// TwinCAT 3 PLC project PLC_IotBase_Test
// ProgramVersion: 3.1.4020.4
// libraries:
//   Tc2_Standard, * (Beckhoff Automation GmbH)
//   Tc2_System, * (Beckhoff Automation GmbH)
//   Tc2_Utilities, * (Beckhoff Automation GmbH)
//   Tc3_DynamicMemory, * (Beckhoff Automation GmbH)
//   Tc3_JsonXml, * (Beckhoff Automation GmbH)
//   Tc3_Module, * (Beckhoff Automation GmbH)
//   Tc3_IotBase,3.1.8.3,Beckhoff Automation GmbH
// project tree:
//   / PlcTask.TcTTO
//   POUs/ FB_TestHTTPLegacy.TcPOU, FB_TestHTTP.TcPOU, FB_TestHTTP_Delete.TcPOU, FB_TestHTTP_Get2.TcPOU, FB_TestHTTP_Trace.TcPOU, FB_TestHTTP_Head.TcPOU, FB_TestHTTP_Connect.TcPOU, FB_TestHTTP_Post.TcPOU, FB_TestHTTP_Get.TcPOU, FB_TestHTTP_Put.TcPOU, FB_TestHTTP_Patch.TcPOU, FB_TestHTTP_Options.TcPOU, FB_TestMqtt.TcPOU, MAIN.TcPOU
// real-time tasks:
//   TASK PlcTask: cycle T#10ms, priority 20, ADS port 350

CONFIGURATION PLC_IotBase_Test
    RESOURCE PLC ON TwinCAT3
        TASK PlcTask(INTERVAL := T#10ms, PRIORITY := 20);
        PROGRAM MAIN WITH PlcTask : MAIN;
    END_RESOURCE
END_CONFIGURATION

// ---- POUs/MAIN.TcPOU
PROGRAM MAIN
VAR
	i : INT;
	bTestMqtt : BOOL;
	fbMqtt : FB_TestMqtt;
	bTestHttp : BOOL := TRUE;
	fbHttp : FB_TestHTTP;
	
END_VAR

i := i + 1;

IF bTestMqtt THEN
	fbMqtt();	
END_IF
IF bTestHttp THEN
	fbHttp();	
END_IF

END_PROGRAM

// ---- POUs/FB_TestMqtt.TcPOU
{attribute 'c++_compatible'}
FUNCTION_BLOCK FB_TestMqtt EXTENDS FB_IotMqttClient
VAR
	hrLastErrorCode : HRESULT;
	bGet : BOOL := TRUE;
	bSetParameter : BOOL := TRUE;
	bConnect : BOOL := TRUE;
	bResetQueue : BOOL;
	sWillPayload : STRING := 'Ich bin dann mal weg.';
	
(* publish *)
	i: INT;
	m : USINT;
	sStr : STRING;
	sTopic1 : STRING(999) := 'test';
	{attribute 'TcEncoding':='UTF-8'}
	sPayload1Wr : STRING := 'Hello world!'; // := STRINGLITERAL_TO_UTF8('Hello world! (üöä)');
	sTopic2 : STRING(999) := '123456789012345678901234567890123456789012345678901234567890123456789012345678901234567890'; // 90 character long
	{attribute 'TcEncoding':='UTF-8'}
	sPayload2Wr : STRING := 'too long?';

(* subscribe *)
	bSubscribed: BOOL;
	{attribute 'TcEncoding':='UTF-8'}
	sPayload1Rd : STRING;
	{attribute 'TcEncoding':='UTF-8'}
	sPayload2Rd : STRING;
	sLastTopic : T_MaxString;
	fbMessageQueue : FB_IotMqttMessageQueue;
	fbMessage : FB_IotMqttMessage;
END_VAR

IF bSetParameter THEN
	bSetParameter := FALSE;
//	SUPER^.sClientId := 'MyTcMqttClient';
	SUPER^.sTopicPrefix := '';
//	SUPER^.sHostName := '172.17.62.85'; //'ba-tradeshows.cloudapp.net', // 'iot.beckhoff.com';
	SUPER^.nHostPort := 1883;
	SUPER^.sUserName := '';
	SUPER^.sUserPassword := '';
	SUPER^.sTopicPrefix := '';
	SUPER^.stTLS.sCA := ''; 
	SUPER^.nKeepAlive := 5;
	
	SUPER^.stWill.sTopic := 'test';
	SUPER^.stWill.pPayload := ADR(sWillPayload);
	SUPER^.stWill.nPayloadSize :=  LEN2(ADR(sWillPayload))+1;
(*
	SUPER^.sTopicPrefix := '';
	SUPER^.sHostName := 'ba-messagebroker.westeurope.cloudapp.azure.com'; // 'localhost'; //'ba-tradeshows.cloudapp.net', // 'iot.beckhoff.com';
	SUPER^.nHostPort := 8883; // 1883;
	SUPER^.sUserName := 'IotAnalytics';
	SUPER^.sUserPassword := '123456';
	SUPER^.sTopicPrefix := 'Beckhoff/Internal/IotAnalytics/';
	SUPER^.stTLS.sCA := 'C:\Projects\IotComm\CA\ca.crt'; // ''; 
*)
	SUPER^.ipMessageQueue := fbMessageQueue;
END_IF

Execute(bConnect);
IF bError THEN
	hrLastErrorCode := hrErrorCode;
END_IF

IF eConnectionState <> ETcIotMqttClientState.MQTT_ERR_NO_CONN THEN
	bConnected := bConnected; // for debugging purposes
END_IF

IF fbMessageQueue.nQueuedMessages > 0 AND bGet THEN
	IF fbMessageQueue.Dequeue(fbMessage) THEN
		IF fbMessage.CompareTopic(sTopic1) THEN
			fbMessage.GetPayload(ADR(sPayload1Rd), SIZEOF(sPayload1Rd), FALSE);
		ELSIF fbMessage.CompareTopic(sTopic2) THEN
			fbMessage.GetPayload(ADR(sPayload2Rd), SIZEOF(sPayload2Rd), FALSE);
		END_IF
	END_IF
END_IF

IF bResetQueue THEN
	bResetQueue := FALSE;
	fbMessageQueue.ResetQueue();
END_IF

IF bConnected THEN
	// subscrive
	IF NOT bSubscribed THEN
		IF Subscribe(sTopic1, 0) AND Subscribe(sTopic2, 0) THEN
			bSubscribed := TRUE;
		ELSE
			hrLastErrorCode := hrErrorCode;
		END_IF
	END_IF
	
	// publish
	i := i + 1;
	IF i = 100 THEN
		m := m + 1;
		sStr := CONCAT('Hello World! (üöä) - ', INT_TO_STRING(m));
		STRING_TO_UTF8(ADR(sPayload1Wr), ADR(sStr), SIZEOF(sPayload1Wr) );
		Publish(sTopic1, ADR(sPayload1Wr), INT_TO_UDINT(LEN(sPayload1Wr)+1), TcIotMqttQos.ExactlyOnceDelivery, FALSE, FALSE);
		IF bError THEN
			hrLastErrorCode := hrErrorCode;
		END_IF
	ELSIF i = 200 THEN
		sPayload1Wr := 'All right?';
		Publish(sTopic1, ADR(sPayload1Wr), INT_TO_UDINT(LEN(sPayload1Wr)+1), 0, FALSE, FALSE);
		IF bError THEN
			hrLastErrorCode := hrErrorCode;
		END_IF
		Publish(sTopic2, ADR(sPayload2Wr), INT_TO_UDINT(LEN(sPayload2Wr)+1), 0, FALSE, FALSE);
		IF bError THEN
			hrLastErrorCode := hrErrorCode;
		END_IF
		i := 0;
	END_IF	
END_IF

{attribute 'c++_compatible'}
{attribute 'signature_flag' := '33554688'}
{attribute 'pack_mode' := '4'}
{attribute 'show'}
{attribute 'minimal_input_size' := '4'}
{attribute 'checksuperglobal'}
METHOD OnMqttMessage : HRESULT
VAR_IN_OUT CONSTANT
	topic	: STRING;
END_VAR
VAR_INPUT
	payload	: PVOID;
	length	: UDINT;
	qos	: TcIotMqttQos;
	repeated	: BOOL;
END_VAR
nMessagesRcv := nMessagesRcv + 1;

STRNCPY( ADR(sLastTopic), ADR(topic), SIZEOF(sLastTopic) );

IF sLastTopic = CONCAT(SUPER^.sTopicPrefix, sTopic1) THEN
	MEMCPY(ADR(sPayload1Rd), payload, MIN(length, DINT_TO_UDINT(SIZEOF(sPayload1Rd))));
ELSIF sLastTopic = CONCAT(SUPER^.sTopicPrefix, sTopic2) THEN
	MEMCPY(ADR(sPayload2Rd), payload, MIN(length, DINT_TO_UDINT(SIZEOF(sPayload2Rd))));
END_IF

OnMqttMessage := S_OK;
END_METHOD

END_FUNCTION_BLOCK

// ---- POUs/FB_TestHTTP.TcPOU
FUNCTION_BLOCK FB_TestHTTP
VAR
	fbClient : FB_IotHttpClient;
	fbRequest: FB_IotHttpRequest;
	fbHeader: FB_IotHttpHeaderFieldMap;
	state : UDINT;
	timeout : UDINT :=10000;
	port : UINT:= 443;
		
	//http://jsonplaceholder.typicode.com/todos/1
	sHostName  : STRING(255) :='jsonplaceholder.typicode.com';
	sCA : STRING(255) := ''; // 'C:\TwinCAT\3.1\Target\Certificates\cloudflare.cer' tls vesrion 1.3 not supported

	fbMqtt_Post: FB_TestHTTP_Post;
	fbMqtt_Get: FB_TestHTTP_Get;
	fbMqtt_Get2: FB_TestHTTP_Get2;	
	fbMqtt_Put: FB_TestHTTP_Put;
	fbMqtt_Patch: FB_TestHTTP_Patch;
	fbMqtt_Trace: FB_TestHTTP_Trace;	
	fbMqtt_Head: FB_TestHTTP_Head;
	fbMqtt_Options: FB_TestHTTP_Options;
	fbMqtt_Delete: FB_TestHTTP_Delete;
	fbMqtt_Connect: FB_TestHTTP_Connect;			
END_VAR

CASE state OF
0:
	fbClient.nConnectTimeout := timeout;
	fbClient.sHostName := sHostName;
	fbClient.bKeepAlive := TRUE;
	IF LEN(STR:=sCA) = 0 THEN
		port:= 80;	
	END_IF
	fbClient.nHostPort := port;
	IF port = 443 THEN
		fbClient.stTLS.sCA :=  sCA;
	END_IF			
	fbHeader.AddField(sField:='MyField', sValue:='MyFieldValue', bAppendValue:= FALSE);
	IF fbClient.bConfigured THEN
		fbClient.Disconnect();
	END_IF	 
	state:=1;
1:	
	IF fbClient.bConfigured THEN 
		fbMqtt_Get(fbClient:=fbClient);
		fbMqtt_Get2(fbClient:=fbClient);
		fbMqtt_Post(fbClient:=fbClient);
		fbMqtt_Put(fbClient:=fbClient);
		fbMqtt_Patch(fbClient:=fbClient);
		fbMqtt_Trace(fbClient:=fbClient);
		fbMqtt_Head(fbClient:=fbClient);
		fbMqtt_Options(fbClient:=fbClient);
		fbMqtt_Delete(fbClient:=fbClient);
		fbMqtt_Connect(fbClient:=fbClient);
	END_IF  	
END_CASE
fbClient.Execute();

END_FUNCTION_BLOCK

// ---- POUs/FB_TestHTTP_Post.TcPOU
FUNCTION_BLOCK FB_TestHTTP_Post
VAR_INPUT
	fbClient : REFERENCE TO FB_IotHttpClient;
END_VAR
VAR	
	fbRequest: FB_IotHttpRequest;
	fbJson: FB_JsonDomParser;
	bSend : BOOL;
	bContinuous : BOOL;
	state : UDINT;
	
	RisingEdge		: R_TRIG;
	sJson: STRING(1024);
	sContent: STRING(1024);	
	
	bJsonRes : BOOL;
	jsonDoc    : SJsonValue;
	jsonVal    : SJsonValue;
		
	reqCount : UDINT;		
	invResCount : UDINT := 0;
	invResValCount : UDINT := 0;
	resVal:STRING;
	nResCnt : UDINT;
	nErrCnt1 : UDINT;
	nErrCnt2 : UDINT;
		
	valOkCount: UDINT;
	
	//http://jsonplaceholder.typicode.com/todos/1
	sUri: STRING(255) := '/posts';
	eRequestType : ETcIotHttpRequestType := ETcIotHttpRequestType.HTTP_POST;		
END_VAR

RisingEdge( CLK:= bSend );
CASE state OF
0:		
	IF fbClient.bConfigured AND (RisingEdge.Q OR bContinuous) THEN 
		fbJson.NewDocument();
		jsonDoc := fbJson.GetDocumentRoot();
		fbJson.AddStringMember(jsonDoc, 'title', 'test1');
		fbJson.AddStringMember(jsonDoc, 'body', 'test2');
		fbJson.AddUintMember(jsonDoc, 'userId', reqCount);
		IF fbRequest.SendJsonDomRequest(sUri:=sUri, fbClient:=fbClient, eRequestType:=eRequestType, fbJson, 0) THEN				
			state := 1;
			reqCount:=reqCount+1;
		END_IF					
	END_IF
1:
	IF NOT fbRequest.bBusy THEN
			IF NOT fbRequest.bError THEN				 
				jsonDoc := fbRequest.GetJsonDomContent(fbJson);				
				IF  jsonDoc <> 0 THEN
					bJsonRes := TRUE;
					fbJson.CopyDocument(sJson, SIZEOF(sJson));
				ELSE
					bJsonRes := FALSE;
				END_IF					
				fbRequest.GetContent(pContent:=ADR(sContent), nContentSize:=SIZEOF(sContent), bSetNullTermination:=TRUE);	
				IF fbRequest.nStatusCode >= 200 AND fbRequest.nStatusCode < 300 THEN
					IF bJsonRes THEN
						IF fbJson.HasMember(jsonDoc, 'userId')  THEN
							jsonVal := fbJson.FindMember(jsonDoc, 'userId');
							IF fbJson.GetUint(jsonVal)+1 = reqCount THEN
								valOkCount:=valOkCount+1;
							ELSE
								invResValCount:=invResValCount+1;
							END_IF
						ELSE 
							invResCount:=invResCount+1;	
						END_IF
					ELSE
						invResCount:=invResCount+1;
					END_IF					
					nResCnt:=nResCnt+1;
				ELSE
					nErrCnt1:=nErrCnt1+1;					
				END_IF				
			ELSE
				nErrCnt2:=nErrCnt2+1;
			END_IF
			state :=0;				
	END_IF  	
END_CASE
fbClient.Execute();

END_FUNCTION_BLOCK

// ---- POUs/FB_TestHTTP_Get.TcPOU
FUNCTION_BLOCK FB_TestHTTP_Get
VAR_INPUT
	fbClient : REFERENCE TO FB_IotHttpClient;
END_VAR
VAR
	
	fbRequest: FB_IotHttpRequest;
	fbJson: FB_JsonDomParser;
	bSend : BOOL;
	bContinuous : BOOL;
	state : UDINT;
	
	RisingEdge		: R_TRIG;
	
	sJson: STRING(300);		
	sContent1: STRING(291);
	bGetContent1 : BOOL;
	nContent1 : UDINT;
	
	bJsonRes : BOOL;
	jsonDoc    : SJsonValue;
	jsonVal    : SJsonValue;
		
	reqCount : UDINT;		
	invResCount : UDINT := 0;
	invResValCount : UDINT := 0;
	resVal:STRING;
	nResCnt : UDINT;
	nErrCnt1 : UDINT;
	nErrCnt2 : UDINT;
		
	valOkCount: UDINT;	
	
	sUri: STRING(255) := '/posts';
	eRequestType : ETcIotHttpRequestType := ETcIotHttpRequestType.HTTP_Get;		
END_VAR

RisingEdge( CLK:= bSend );
CASE state OF
0:	
	IF fbClient.bConfigured AND (RisingEdge.Q OR bContinuous) THEN 
		IF fbRequest.SendRequest(sUri:=sUri, fbClient:=fbClient, eRequestType:=eRequestType, 0, 0, 0) THEN				
			state := 1;
			reqCount:=reqCount+1;
		END_IF					
	END_IF
1:
	IF NOT fbRequest.bBusy THEN
			IF NOT fbRequest.bError THEN				 
				jsonDoc := fbRequest.GetJsonDomContent(fbJson);
				IF  jsonDoc <> 0 THEN
					bJsonRes := TRUE;
					fbJson.CopyDocument(sJson, SIZEOF(sJson)-1);
				ELSE
					bJsonRes := FALSE;
				END_IF					
				bGetContent1 := fbRequest.GetContent(pContent:=ADR(sContent1), nContentSize:=SIZEOF(sContent1), bSetNullTermination:=TRUE);
				nContent1:= LEN2(ADR(sContent1));
				IF fbRequest.nStatusCode >= 200 AND fbRequest.nStatusCode < 300 THEN
					IF bJsonRes THEN													 								
						IF fbJson.IsArray(jsonDoc) AND fbJson.GetArraySize(jsonDoc) > 0 THEN
							jsonVal := fbJson.GetArrayValueByIdx(jsonDoc, 0);
							IF fbJson.HasMember(jsonVal, 'id')  THEN							
								jsonVal := fbJson.FindMember(jsonVal, 'id');
								IF fbJson.GetUint(jsonVal) = 1 THEN
									valOkCount:=valOkCount+1;
								ELSE
									invResValCount:=invResValCount+1;
								END_IF
							ELSE 
								invResCount:=invResCount+1;	
						END_IF
						ELSE 
							invResCount:=invResCount+1;	
						END_IF
					ELSE
						invResCount:=invResCount+1;
					END_IF					
					nResCnt:=nResCnt+1;
				ELSE
					nErrCnt1:=nErrCnt1+1;					
				END_IF				
			ELSE
				nErrCnt2:=nErrCnt2+1;
			END_IF
			state :=0;				
	END_IF  	
END_CASE
fbClient.Execute();

END_FUNCTION_BLOCK

// ---- POUs/FB_TestHTTP_Get2.TcPOU
FUNCTION_BLOCK FB_TestHTTP_Get2 (*checks GetContent *)
VAR_INPUT
	fbClient : REFERENCE TO FB_IotHttpClient;
END_VAR
VAR
	
	fbRequest: FB_IotHttpRequest;
	fbJson: FB_JsonDomParser;
	bSend : BOOL;
	bContinuous : BOOL;
	state : UDINT;
	
	RisingEdge		: R_TRIG;
	
	sJson: STRING(300);
	
	bGetContent1 : BOOL;
	bGetContent2 : BOOL;
	bGetContent3 : BOOL;
	bGetContent4 : BOOL;
	bGetContent5 : BOOL;					
	sContent1: STRING(291);
	sContent2: STRING(292);
	sContent3: STRING(293);	
	sContent4: STRING(5);
	sContent5: STRING(300) := '123456789012345678901234567890123456789012345678901234567890123456789012345678901234567890123456789x123456789012345678901234567890123456789012345678901234567890123456789012345678901234567890123456789x123456789012345678901234567890123456789012345678901234567890123456789012345678901234567890123456789x';
	sTest:String := '123';
	nContent1: UDINT;
	nContent2: UDINT;
	nContent3: UDINT;
	nContent4: UDINT;
	nFind1:UDINT;
	nFind2:UDINT;
	nFind3:UDINT;
	nFind4:UDINT;
	nFind5:UDINT;
	nLenT1:UDINT;
	nLen2T1:INT;
	sT1: STRING(3) :='123';
	
	sServer: STRING(10) := 'cloudflare';
	sServer1: STRING(9);
	sServer2: STRING(10);
	sServer3: STRING(11);
	lenSrv1 : UDINT;
	lenSrv2 : UDINT;
	lenSrv3 : UDINT;
	findSrv1 : UDINT;
	findSrv2 : UDINT;
	findSrv3 : UDINT;
	findSrv4 : UDINT;
	bGetSrv1: BOOL;
	bGetSrv2: BOOL;	
	bGetSrv3: BOOL;
	
	
	
	nSizeT1 : UDINT; 
	testCnt1:UDINT;
	testCnt2:UDINT;
	
	bJsonRes : BOOL;
	jsonDoc    : SJsonValue;
	jsonVal    : SJsonValue;
		
	reqCount : UDINT;		
	invResCount : UDINT := 0;
	invResValCount : UDINT := 0;
	resVal:STRING;
	nResCnt : UDINT;
	nErrCnt1 : UDINT;
	nErrCnt2 : UDINT;
	nErrCnt3 : UDINT;
	nErrCnt4 : UDINT;
		
	valOkCount: UDINT;	
	
	sUri: STRING(255) := '/posts/1';
	eRequestType : ETcIotHttpRequestType := ETcIotHttpRequestType.HTTP_Get;	
	sContent: INT;
	
	pByte : POINTER TO BYTE;
	pUdint : POINTER TO UDINT;
	t: UDINT:=0;	
END_VAR

RisingEdge( CLK:= bSend );
CASE state OF
0:	
	IF fbClient.bConfigured AND ( (t=1) OR (RisingEdge.Q OR bContinuous)) THEN
		IF t = 2 THEN
			t:=0;
		END_IF 
		IF fbRequest.SendRequest(sUri:=sUri, fbClient:=fbClient, eRequestType:=eRequestType, 0, 0, 0) THEN				
			state := 1;
			reqCount:=reqCount+1;			
		END_IF					
	END_IF
1:
	IF NOT fbRequest.bBusy THEN
			IF NOT fbRequest.bError THEN				 
				jsonDoc := fbRequest.GetJsonDomContent(fbJson);
				IF  jsonDoc <> 0 THEN
					bJsonRes := TRUE;
					fbJson.CopyDocument(sJson, SIZEOF(sJson)-1);
				ELSE
					bJsonRes := FALSE;
				END_IF					
				
				(*
					HttpClient always appends 0(not included in content length) and Http Responses normally don't include 0
					so to test content with an appended 0 one has to patch content lenght of response
				*)
				IF t = 0 THEN
					pByte :=  fbRequest.pContent+fbRequest.nContentSize-1;
					IF pByte^ <> 0 THEN					
						pByte :=  fbRequest.pContent+fbRequest.nContentSize;
						IF pByte^ = 0 THEN
							pByte :=  fbRequest.pContent+fbRequest.nContentSize-1;
							pUdint := ADR(fbRequest.nContentSize); 
							pUdint^:=fbRequest.nContentSize+1;
							testCnt1:=testCnt1+1;
						END_IF						
					END_IF
					t:=1;
				ELSE
					testCnt2:=testCnt2+1;
					t:=2;
				END_IF
				
				bGetContent1 := fbRequest.GetContent(pContent:=ADR(sContent1), nContentSize:=SIZEOF(sContent1), bSetNullTermination:=TRUE);
				bGetContent2 := fbRequest.GetContent(pContent:=ADR(sContent2), nContentSize:=SIZEOF(sContent2), bSetNullTermination:=TRUE);
				bGetContent3 := fbRequest.GetContent(pContent:=ADR(sContent3), nContentSize:=SIZEOF(sContent3), bSetNullTermination:=TRUE);
				bGetContent4 := fbRequest.GetContent(pContent:=ADR(sContent4), nContentSize:=SIZEOF(sContent4), bSetNullTermination:=TRUE);
				bGetContent5 := fbRequest.GetContent(pContent:=ADR(sContent5), nContentSize:=SIZEOF(sContent5), bSetNullTermination:=TRUE);
				nContent1 := LEN2(ADR(sContent1));
				nContent2 := LEN2(ADR(sContent2));
				nContent3 := LEN2(ADR(sContent3));
				nContent4 := LEN2(ADR(sContent4));
				nFind1:= FIND2(ADR(sContent2), ADR(sContent3));
				nFind2:= FIND2(ADR(sContent2), ADR(sContent1));
				nFind3:= FIND2(ADR(sContent1), ADR(sContent2));
				nFind4:= FIND2(ADR(sContent2), ADR(sContent4));
				nFind5:= FIND2(ADR(sContent3), ADR(sContent5));
				nLenT1:=LEN2(ADR(sT1));
				nLen2T1:=LEN(sT1);
				nSizeT1:=SIZEOF(sT1);												
				
				IF NOT (bGetContent1 = FALSE AND bGetContent2 = TRUE AND bGetContent3 = TRUE AND bGetContent4 = FALSE AND nFind1=1 AND nFind2=1 AND nFind3=0 AND nFind4=1 AND nFind5=1 AND nContent1 = 291 AND nContent2 = 292 AND nContent3 = 292 AND nContent4 = 5)  THEN
					nErrCnt3:=nErrCnt3+1;
				END_IF				
				
				bGetSrv1 := fbRequest.GetHeaderField('server', ADR(sServer1), SIZEOF(sServer1));
				bGetSrv2 := fbRequest.GetHeaderField('server', ADR(sServer2), SIZEOF(sServer2));
				bGetSrv3 := fbRequest.GetHeaderField('server', ADR(sServer3), SIZEOF(sServer3));
				lenSrv1 := LEN2(ADR(sServer1));
				lenSrv2 := LEN2(ADR(sServer2));
				lenSrv3 := LEN2(ADR(sServer3));
				findSrv1:= FIND2(ADR(sServer2), ADR(sServer3));
				findSrv2:= FIND2(ADR(sServer2), ADR(sServer1));
				findSrv3:= FIND2(ADR(sServer1), ADR(sServer2));
				findSrv4:= FIND2(ADR(sServer), ADR(sServer2));
				
				IF NOT (bGetSrv1 = FALSE AND bGetSrv2 = TRUE AND lenSrv1 = 9 AND lenSrv2 = 10 AND lenSrv3 = 10 AND findSrv1 = 1 AND findSrv2 = 1 AND findSrv3 = 0 AND findSrv4=1 ) THEN
					nErrCnt4:=nErrCnt4+1;
				END_IF 

				IF fbRequest.nStatusCode >= 200 AND fbRequest.nStatusCode < 300 THEN
					IF bJsonRes THEN													 								
						IF fbJson.HasMember(jsonDoc, 'id')  THEN							
							jsonVal := fbJson.FindMember(jsonDoc, 'id');
							IF fbJson.GetUint(jsonVal) = 1 THEN
								valOkCount:=valOkCount+1;
							ELSE
								invResValCount:=invResValCount+1;
							END_IF
						ELSE 
							invResCount:=invResCount+1;	
						END_IF						
					ELSE
						invResCount:=invResCount+1;
					END_IF					
					nResCnt:=nResCnt+1;
				ELSE
					nErrCnt1:=nErrCnt1+1;					
				END_IF
					
			ELSE
				nErrCnt2:=nErrCnt2+1;
			END_IF
			state :=0;				
	END_IF  	
END_CASE
fbClient.Execute();

END_FUNCTION_BLOCK

// ---- POUs/FB_TestHTTP_Put.TcPOU
FUNCTION_BLOCK FB_TestHTTP_Put
VAR_INPUT
	fbClient : REFERENCE TO FB_IotHttpClient;
END_VAR
VAR	
	fbRequest: FB_IotHttpRequest;
	fbJson: FB_JsonDomParser;
	bSend : BOOL;
	bContinuous : BOOL;
	state : UDINT;
	
	RisingEdge		: R_TRIG;
	sJson: STRING(1024);
sContent: STRING(1024);	
	
	bJsonRes : BOOL;
	jsonDoc    : SJsonValue;
	jsonVal    : SJsonValue;
		
	reqCount : UDINT;		
	invResCount : UDINT := 0;
	invResValCount : UDINT := 0;
	resVal:STRING;
	nResCnt : UDINT;
	nErrCnt1 : UDINT;
	nErrCnt2 : UDINT;
		
	valOkCount: UDINT;
	
	//http://jsonplaceholder.typicode.com/todos/1
	sUri: STRING(255) := '/posts/1';
	eRequestType : ETcIotHttpRequestType := ETcIotHttpRequestType.HTTP_Put;		
END_VAR

RisingEdge( CLK:= bSend );
CASE state OF
0:		
	IF fbClient.bConfigured AND (RisingEdge.Q OR bContinuous) THEN 
		fbJson.NewDocument();
		jsonDoc := fbJson.GetDocumentRoot();
		fbJson.AddStringMember(jsonDoc, 'id', '1');
		fbJson.AddStringMember(jsonDoc, 'title', 'test1');
		fbJson.AddStringMember(jsonDoc, 'body', 'test2');
		fbJson.AddUintMember(jsonDoc, 'userId', reqCount);
		IF fbRequest.SendJsonDomRequest(sUri:=sUri, fbClient:=fbClient, eRequestType:=eRequestType, fbJson, 0) THEN				
			state := 1;
			reqCount:=reqCount+1;
		END_IF					
	END_IF
1:
	IF NOT fbRequest.bBusy THEN
			IF NOT fbRequest.bError THEN				 
				jsonDoc := fbRequest.GetJsonDomContent(fbJson);				
				IF  jsonDoc <> 0 THEN
					bJsonRes := TRUE;
					fbJson.CopyDocument(sJson, SIZEOF(sJson));
				ELSE
					bJsonRes := FALSE;
				END_IF					
				fbRequest.GetContent(pContent:=ADR(sContent), nContentSize:=SIZEOF(sContent), bSetNullTermination:=TRUE);	
				IF fbRequest.nStatusCode >= 200 AND fbRequest.nStatusCode < 300 THEN
					IF bJsonRes THEN
						IF fbJson.HasMember(jsonDoc, 'userId')  THEN
							jsonVal := fbJson.FindMember(jsonDoc, 'userId');
							IF fbJson.GetUint(jsonVal)+1 = reqCount THEN
								valOkCount:=valOkCount+1;
							ELSE
								invResValCount:=invResValCount+1;
							END_IF
						ELSE 
							invResCount:=invResCount+1;	
						END_IF
					ELSE
						invResCount:=invResCount+1;
					END_IF					
					nResCnt:=nResCnt+1;
				ELSE
					nErrCnt1:=nErrCnt1+1;					
				END_IF				
			ELSE
				nErrCnt2:=nErrCnt2+1;
			END_IF
			state :=0;				
	END_IF  	
END_CASE
fbClient.Execute();

END_FUNCTION_BLOCK

// ---- POUs/FB_TestHTTP_Patch.TcPOU
FUNCTION_BLOCK FB_TestHTTP_Patch
VAR_INPUT
	fbClient : REFERENCE TO FB_IotHttpClient;
END_VAR
VAR	
	fbRequest: FB_IotHttpRequest;
	fbJson: FB_JsonDomParser;
	bSend : BOOL;
	bContinuous : BOOL;
	state : UDINT;
	
	RisingEdge		: R_TRIG;
	sJson: STRING(1024);
	sContent: STRING(1024);	
	
	bJsonRes : BOOL;
	jsonDoc    : SJsonValue;
	jsonVal    : SJsonValue;
		
	reqCount : UDINT;		
	invResCount : UDINT := 0;
	invResValCount : UDINT := 0;
	resVal:STRING;
	nResCnt : UDINT;
	nErrCnt1 : UDINT;
	nErrCnt2 : UDINT;
		
	valOkCount: UDINT;
	
	//http://jsonplaceholder.typicode.com/todos/1
	sUri: STRING(255) := '/posts/1';
	eRequestType : ETcIotHttpRequestType := ETcIotHttpRequestType.HTTP_Patch;		
END_VAR

RisingEdge( CLK:= bSend );
CASE state OF
0:		
	IF fbClient.bConfigured AND (RisingEdge.Q OR bContinuous) THEN 
		fbJson.NewDocument();
		jsonDoc := fbJson.GetDocumentRoot();
		fbJson.AddUintMember(jsonDoc, 'title', reqCount);
		IF fbRequest.SendJsonDomRequest(sUri:=sUri, fbClient:=fbClient, eRequestType:=eRequestType, fbJson, 0) THEN				
			state := 1;
			reqCount:=reqCount+1;
		END_IF					
	END_IF
1:
	IF NOT fbRequest.bBusy THEN
			IF NOT fbRequest.bError THEN				 
				jsonDoc := fbRequest.GetJsonDomContent(fbJson);				
				IF  jsonDoc <> 0 THEN
					bJsonRes := TRUE;
					fbJson.CopyDocument(sJson, SIZEOF(sJson));
				ELSE
					bJsonRes := FALSE;
				END_IF					
				fbRequest.GetContent(pContent:=ADR(sContent), nContentSize:=SIZEOF(sContent), bSetNullTermination:=TRUE);	
				IF fbRequest.nStatusCode >= 200 AND fbRequest.nStatusCode < 300 THEN
					IF bJsonRes THEN
						IF fbJson.HasMember(jsonDoc, 'title')  THEN
							jsonVal := fbJson.FindMember(jsonDoc, 'title');
							IF fbJson.GetUint(jsonVal)+1 = reqCount THEN
								valOkCount:=valOkCount+1;
							ELSE
								invResValCount:=invResValCount+1;
							END_IF
						ELSE 
							invResCount:=invResCount+1;	
						END_IF
					ELSE
						invResCount:=invResCount+1;
					END_IF					
					nResCnt:=nResCnt+1;
				ELSE
					nErrCnt1:=nErrCnt1+1;					
				END_IF				
			ELSE
				nErrCnt2:=nErrCnt2+1;
			END_IF
			state :=0;				
	END_IF  	
END_CASE
fbClient.Execute();

END_FUNCTION_BLOCK

// ---- POUs/FB_TestHTTP_Trace.TcPOU
FUNCTION_BLOCK FB_TestHTTP_Trace
VAR_INPUT
	fbClient : REFERENCE TO FB_IotHttpClient;
END_VAR
VAR
	
	fbRequest: FB_IotHttpRequest;
	fbJson: FB_JsonDomParser;
	bSend : BOOL;
	bContinuous : BOOL;
	state : UDINT;
	
	RisingEdge		: R_TRIG;
	
	sJson: STRING(1024);		
	sContent: STRING(1024);
	
	bJsonRes : BOOL;
	jsonDoc    : SJsonValue;
	jsonVal    : SJsonValue;
		
	reqCount : UDINT;		
	invResCount : UDINT := 0;
	invResValCount : UDINT := 0;
	resVal:STRING;
	nResCnt : UDINT;
	nErrCnt1 : UDINT;
	nErrCnt2 : UDINT;
		
	valOkCount: UDINT;	
	
	sUri: STRING(255) := '/posts';
	eRequestType : ETcIotHttpRequestType := ETcIotHttpRequestType.HTTP_TRACE;	
END_VAR

RisingEdge( CLK:= bSend );
CASE state OF
0:	
	IF fbClient.bConfigured AND (RisingEdge.Q OR bContinuous) THEN 
		IF fbRequest.SendRequest(sUri:=sUri, fbClient:=fbClient, eRequestType:=eRequestType, 0, 0, 0) THEN				
			state := 1;
			reqCount:=reqCount+1;
		END_IF					
	END_IF
1:
	IF NOT fbRequest.bBusy THEN
			IF NOT fbRequest.bError THEN				 
				jsonDoc := fbRequest.GetJsonDomContent(fbJson);
				IF  jsonDoc <> 0 THEN
					bJsonRes := TRUE;
					fbJson.CopyDocument(sJson, SIZEOF(sJson)-1);
				ELSE
					bJsonRes := FALSE;
				END_IF					
				fbRequest.GetContent(pContent:=ADR(sContent), nContentSize:=SIZEOF(sContent), bSetNullTermination:=TRUE);	
				IF fbRequest.nStatusCode >= 200 AND fbRequest.nStatusCode < 300 THEN
					IF bJsonRes THEN													 								
						IF fbJson.IsArray(jsonDoc) AND fbJson.GetArraySize(jsonDoc) > 0 THEN
							jsonVal := fbJson.GetArrayValueByIdx(jsonDoc, 0);
							IF fbJson.HasMember(jsonVal, 'id')  THEN							
								jsonVal := fbJson.FindMember(jsonVal, 'id');
								IF fbJson.GetUint(jsonVal) = 1 THEN
									valOkCount:=valOkCount+1;
								ELSE
									invResValCount:=invResValCount+1;
								END_IF
							ELSE 
								invResCount:=invResCount+1;	
						END_IF
						ELSE 
							invResCount:=invResCount+1;	
						END_IF
					ELSE
						invResCount:=invResCount+1;
					END_IF					
					nResCnt:=nResCnt+1;
				ELSE
					nErrCnt1:=nErrCnt1+1;					
				END_IF				
			ELSE
				nErrCnt2:=nErrCnt2+1;
			END_IF
			state :=0;				
	END_IF  	
END_CASE
fbClient.Execute();

END_FUNCTION_BLOCK

// ---- POUs/FB_TestHTTP_Head.TcPOU
FUNCTION_BLOCK FB_TestHTTP_Head
VAR_INPUT
	fbClient : REFERENCE TO FB_IotHttpClient;
END_VAR
VAR	
	fbRequest: FB_IotHttpRequest;
	fbJson: FB_JsonDomParser;
	bSend : BOOL;
	bContinuous : BOOL;
	state : UDINT;
	
	RisingEdge		: R_TRIG;	
	sContentLen: STRING(256);	
	
	bJsonRes : BOOL;
	jsonDoc    : SJsonValue;
	jsonVal    : SJsonValue;
		
	reqCount : UDINT;		
	invResCount : UDINT := 0;
	invResValCount : UDINT := 0;
	resVal:STRING;
	nResCnt : UDINT;
	nErrCnt1 : UDINT;
	nErrCnt2 : UDINT;
		
	valOkCount: UDINT;
	
	//http://jsonplaceholder.typicode.com/todos/1
	sUri: STRING(255) := '/posts/1';
	eRequestType : ETcIotHttpRequestType := ETcIotHttpRequestType.HTTP_HEAD;		
END_VAR

RisingEdge( CLK:= bSend );
CASE state OF
0:		
	IF fbClient.bConfigured AND (RisingEdge.Q OR bContinuous) THEN 
		IF fbRequest.SendRequest(sUri:=sUri, fbClient:=fbClient, eRequestType:=eRequestType, 0, 0, 0) THEN				
			state := 1;
			reqCount:=reqCount+1;
		END_IF					
	END_IF
1:
	IF NOT fbRequest.bBusy THEN
			IF NOT fbRequest.bError THEN				 
				IF fbRequest.GetHeaderField('Content-Length', ADR(sContentLen), SIZEOF(sContentLen)) THEN 
					IF STRING_TO_UDINT(sContentLen) = 292 THEN
						valOkCount:=valOkCount+1;
					ELSE
						invResValCount:=invResValCount+1;
					END_IF
				ELSE
					invResCount:=invResCount+1;
				END_IF
			ELSE
				nErrCnt2:=nErrCnt2+1;
			END_IF
			state :=0;				
	END_IF  	
END_CASE
fbClient.Execute();

END_FUNCTION_BLOCK

// ---- POUs/FB_TestHTTP_Options.TcPOU
FUNCTION_BLOCK FB_TestHTTP_Options
VAR_INPUT
	fbClient : REFERENCE TO FB_IotHttpClient;
END_VAR
VAR
	
	fbRequest: FB_IotHttpRequest;
	fbJson: FB_JsonDomParser;
	bSend : BOOL;
	bContinuous : BOOL;
	state : UDINT;
	
	RisingEdge		: R_TRIG;
	
	sJson: STRING(1024);		
	sContent: STRING(1024);
	sAllow: STRING(100);
	
	bJsonRes : BOOL;
	jsonDoc    : SJsonValue;
	jsonVal    : SJsonValue;
		
	reqCount : UDINT;		
	invResCount : UDINT := 0;
	invResValCount : UDINT := 0;
	resVal:STRING;
	nResCnt : UDINT;
	nErrCnt1 : UDINT;
	nErrCnt2 : UDINT;
		
	valOkCount: UDINT;	
	
	sUri: STRING(255) := '/posts';
	eRequestType : ETcIotHttpRequestType := ETcIotHttpRequestType.HTTP_OPTIONS;		
END_VAR

RisingEdge( CLK:= bSend );
CASE state OF
0:	
	IF fbClient.bConfigured AND (RisingEdge.Q OR bContinuous) THEN 
		IF fbRequest.SendRequest(sUri:=sUri, fbClient:=fbClient, eRequestType:=eRequestType, 0, 0, 0) THEN				
			state := 1;
			reqCount:=reqCount+1;
		END_IF					
	END_IF
1:
	IF NOT fbRequest.bBusy THEN
			IF NOT fbRequest.bError THEN
				//IF f Access-Control-Allow-Methods: GET,HEAD,PUT,PATCH,POST,DELETE				 
				//;
				IF fbRequest.GetHeaderField('Access-Control-Allow-Methods', ADR(sAllow), SIZEOF(sAllow)) THEN 
					IF Find(sAllow, 'POST') <> 0 THEN
						valOkCount:=valOkCount+1;
					ELSE
						invResValCount:=invResValCount+1;
					END_IF
				ELSE
					invResCount:=invResCount+1;
				END_IF								
			ELSE
				nErrCnt2:=nErrCnt2+1;
			END_IF
			state :=0;				
	END_IF  	
END_CASE
fbClient.Execute();

END_FUNCTION_BLOCK

// ---- POUs/FB_TestHTTP_Delete.TcPOU
FUNCTION_BLOCK FB_TestHTTP_Delete
VAR_INPUT
	fbClient : REFERENCE TO FB_IotHttpClient;
END_VAR
VAR	
	fbRequest: FB_IotHttpRequest;
	fbJson: FB_JsonDomParser;
	bSend : BOOL;
	bContinuous : BOOL;
	state : UDINT;
	
	RisingEdge		: R_TRIG;
	sJson: STRING(1024);
	sContent: STRING(1024);	
	
	bJsonRes : BOOL;
	jsonDoc    : SJsonValue;
	jsonVal    : SJsonValue;
		
	reqCount : UDINT;		
	invResCount : UDINT := 0;
	invResValCount : UDINT := 0;
	resVal:STRING;
	nResCnt : UDINT;
	nErrCnt1 : UDINT;
	nErrCnt2 : UDINT;
		
	valOkCount: UDINT;
	
	//http://jsonplaceholder.typicode.com/todos/1
	sUri: STRING(255) := '/posts/2';
	eRequestType : ETcIotHttpRequestType := ETcIotHttpRequestType.HTTP_Delete;		
END_VAR

RisingEdge( CLK:= bSend );
CASE state OF
0:		
	IF fbClient.bConfigured AND (RisingEdge.Q OR bContinuous) THEN 
		IF fbRequest.SendRequest(sUri:=sUri, fbClient:=fbClient, eRequestType:=eRequestType, 0, 0, 0) THEN				
			state := 1;
			reqCount:=reqCount+1;
		END_IF					
	END_IF
1:
	IF NOT fbRequest.bBusy THEN
			IF NOT fbRequest.bError THEN				 
				jsonDoc := fbRequest.GetJsonDomContent(fbJson);				
				IF  jsonDoc <> 0 THEN
					bJsonRes := TRUE;
					fbJson.CopyDocument(sJson, SIZEOF(sJson));
				ELSE
					bJsonRes := FALSE;
				END_IF					
				fbRequest.GetContent(pContent:=ADR(sContent), nContentSize:=SIZEOF(sContent), bSetNullTermination:=TRUE);	
				IF fbRequest.nStatusCode >= 200 AND fbRequest.nStatusCode < 300 THEN
					IF bJsonRes THEN
						valOkCount:=valOkCount+1;						
					ELSE
						invResCount:=invResCount+1;
					END_IF					
					nResCnt:=nResCnt+1;
				ELSE
					nErrCnt1:=nErrCnt1+1;					
				END_IF				
			ELSE
				nErrCnt2:=nErrCnt2+1;
			END_IF
			state :=0;				
	END_IF  	
END_CASE
fbClient.Execute();

END_FUNCTION_BLOCK

// ---- POUs/FB_TestHTTP_Connect.TcPOU
FUNCTION_BLOCK FB_TestHTTP_Connect
VAR_INPUT
	fbClient : REFERENCE TO FB_IotHttpClient;
END_VAR
VAR	
	fbRequest: FB_IotHttpRequest;
	fbJson: FB_JsonDomParser;
	bSend : BOOL;
	bContinuous : BOOL;
	state : UDINT;
	
	RisingEdge		: R_TRIG;
	sJson: STRING(1024);
	sContent: STRING(1024);
	
	bJsonRes : BOOL;
	jsonDoc    : SJsonValue;
	jsonVal    : SJsonValue;
		
	reqCount : UDINT;		
	invResCount : UDINT := 0;
	invResValCount : UDINT := 0;
	resVal:STRING;
	nResCnt : UDINT;
	nErrCnt1 : UDINT;
	nErrCnt2 : UDINT;
		
	valOkCount: UDINT;
	
	//http://jsonplaceholder.typicode.com/todos/1
	sUri: STRING(255) := '/posts/1';
	eRequestType : ETcIotHttpRequestType := ETcIotHttpRequestType.HTTP_Connect;		
END_VAR

RisingEdge( CLK:= bSend );
CASE state OF
0:		
	IF fbClient.bConfigured AND (RisingEdge.Q OR bContinuous) THEN 
		IF fbRequest.SendRequest(sUri:=sUri, fbClient:=fbClient, eRequestType:=eRequestType, 0, 0, 0) THEN				
			state := 1;
			reqCount:=reqCount+1;
		END_IF					
	END_IF
1:
	IF NOT fbRequest.bBusy THEN
			IF NOT fbRequest.bError THEN				 
				jsonDoc := fbRequest.GetJsonDomContent(fbJson);				
				IF  jsonDoc <> 0 THEN
					bJsonRes := TRUE;
					fbJson.CopyDocument(sJson, SIZEOF(sJson));
				ELSE
					bJsonRes := FALSE;
				END_IF					
				fbRequest.GetContent(pContent:=ADR(sContent), nContentSize:=SIZEOF(sContent), bSetNullTermination:=TRUE);	
				IF fbRequest.nStatusCode >= 200 AND fbRequest.nStatusCode < 300 THEN
					IF bJsonRes THEN
						IF fbJson.HasMember(jsonDoc, 'title')  THEN
							jsonVal := fbJson.FindMember(jsonDoc, 'title');
							IF fbJson.GetUint(jsonVal)+1 = reqCount THEN
								valOkCount:=valOkCount+1;
							ELSE
								invResValCount:=invResValCount+1;
							END_IF
						ELSE 
							invResCount:=invResCount+1;	
						END_IF
					ELSE
						invResCount:=invResCount+1;
					END_IF					
					nResCnt:=nResCnt+1;
				ELSE
					nErrCnt1:=nErrCnt1+1;					
				END_IF				
			ELSE
				nErrCnt2:=nErrCnt2+1;
			END_IF
			state :=0;				
	END_IF  	
END_CASE
fbClient.Execute();

END_FUNCTION_BLOCK

// ---- POUs/FB_TestHTTPLegacy.TcPOU
FUNCTION_BLOCK FB_TestHTTPLegacy
VAR
	fbClient : FB_IotHttpClient;
	fbRequest: FB_IotHttpRequest;
	bWithHeader : BOOL;
	fbHeader: FB_IotHttpHeaderFieldMap;
	fbJson: FB_JsonDomParser;
	bSend : BOOL;
	bContinuous : BOOL;
	state : UDINT;
	
	nResCnt : UDINT;
	nErrCnt1 : UDINT;
	nErrCnt2 : UDINT;
	RisingEdge		: R_TRIG;
	sContent: STRING(1024);
	sJson: STRING(1024);
	sServer : STRING(255);
	pSndContent : PVOID;
	nSndContent: UDINT;
	port : UINT:= 443;
	reqCount : UDINT;	
	bJsonRes : BOOL;
	jsonDoc    : SJsonValue;
	jsonVal    : SJsonValue;
		timeout : UDINT :=10000;	
	invResCount : UDINT := 0;
	invResValCount : UDINT := 0;
	resVal:STRING;	
	valOkCount: UDINT;	
	(*
	//http://jsonplaceholder.typicode.com/todos/1
	sHostName  : STRING(255) :='jsonplaceholder.typicode.com'
	sUri: STRING(255) := '/todos/1';
	sCA : STRING(255) := ''; // 'C:\TwinCAT\3.1\Target\Certificates\cloudflare.cer' tls vesrion 1.3 not supported	
	eRequestType : ETcIotHttpRequestType := ETcIotHttpRequestType.HTTP_GET;
	sSndContent: STRING(255):='';
	bDynamicContent : BOOL :=FALSE;
	bJson : BOOL:=FALSE;	
	*)
	
	//http://jsonplaceholder.typicode.com/todos/1
	sHostName  : STRING(255) :='jsonplaceholder.typicode.com';
	sUri: STRING(255) := '/posts';
	sCA : STRING(255) := ''; // 'C:\TwinCAT\3.1\Target\Certificates\cloudflare.cer' tls vesrion 1.3 not supported	
	eRequestType : ETcIotHttpRequestType := ETcIotHttpRequestType.HTTP_POST;
	sSndContent: STRING(255):='{"title": "test1", "body": "test2", "userId": 2}';
	bDynamicContent : BOOL :=FALSE;
	bJson : BOOL:=TRUE;
	(*
	//https://postman-echo.com/get?foo1=bar1&foo2=bar2
	sHostName : STRING(255) := 'postman-echo.com';
	sUri: STRING(255) := '/get?foo1=bar1&foo2=bar2'; //	https://postman-echo.com/get?foo1=bar1&foo2=bar2
	sCA : STRING(255) := 'C:\TwinCAT\3.1\Target\Certificates\amazon.cer';
	eRequestType : ETcIotHttpRequestType := ETcIotHttpRequestType.HTTP_GET;
	sSndContent: STRING(255):='';
	bDynamicContent : BOOL :=FALSE;
	bJson : BOOL:=FALSE;
	*)
	
	//https://postman-echo.com/get?foo1=bar1&foo2=bar2
	(*
	sHostName : STRING(255) := 'postman-echo.com';
	sCA : STRING(255) := 'C:\TwinCAT\3.1\Target\Certificates\amazon.cer';
	sUri: STRING(255) := '/post'; //	https://postman-echo.com/post
	eRequestType : ETcIotHttpRequestType := ETcIotHttpRequestType.HTTP_POST;
	bDynamicContent : BOOL :=TRUE;	
	bJson : BOOL:=FALSE;
	sSndContent: STRING(255):='';
	*)
	
	//https://api.openweathermap.org/data/2.5/weather?q=London,uk&APPID=0844c0a29ad58753b478183254b1eb89
	(*sHostName : STRING(255) := 'api.openweathermap.org';
	sUri: STRING(255) := '/data/2.5/weather?q=London,uk&APPID=0844c0a29ad58753b478183254b1eb89';
	sCA : STRING(255) := 'C:\TwinCAT\3.1\Target\Certificates\weathermap.cer';
	eRequestType : ETcIotHttpRequestType := ETcIotHttpRequestType.HTTP_GET;
	sSndContent: STRING(255):='';
	bDynamicContent : BOOL :=FALSE;
	bJson : BOOL:=FALSE;
	*)
	
	(*
	sHostName : STRING(255) := '192.168.1.8';
	sUri: STRING(255) := '/index';
	sCA : STRING(255) := 'C:\TwinCAT\3.1\Target\Certificates\cx9020.cer';
	eRequestType : ETcIotHttpRequestType := ETcIotHttpRequestType.HTTP_GET;
	sSndContent: STRING(255):='';
	bDynamicContent : BOOL :=FALSE;	
	bJson : BOOL:=FALSE;
	*)

END_VAR

RisingEdge( CLK:= bSend );
CASE state OF
0:
	fbClient.nConnectTimeout := timeout;
	fbClient.sHostName := sHostName;
	fbClient.bKeepAlive := TRUE;
	IF LEN(STR:=sCA) = 0 THEN
		port:= 80;	
	END_IF
	fbClient.nHostPort := port;
	IF port = 443 THEN
		fbClient.stTLS.sCA :=  sCA;
	END_IF			
	fbHeader.AddField(sField:='MyField', sValue:='MyFieldValue', bAppendValue:= FALSE);
	IF fbClient.bConfigured THEN
		fbClient.Disconnect();
	END_IF	 
	state:=1;
1:	
	IF fbClient.bConfigured AND (RisingEdge.Q OR bContinuous) THEN 
		sServer:='';
		IF bJson THEN
			fbJson.NewDocument();
			jsonDoc := fbJson.GetDocumentRoot();
			fbJson.AddStringMember(jsonDoc, 'title', 'test1');
			fbJson.AddStringMember(jsonDoc, 'body', 'test2');
			fbJson.AddUintMember(jsonDoc, 'userId', reqCount);
			IF NOT bWithHeader THEN
				IF fbRequest.SendJsonDomRequest(sUri:=sUri, fbClient:=fbClient, eRequestType:=eRequestType, fbJson, 0) THEN				
					state := 2;
					reqCount:=reqCount+1;
				END_IF
			ELSE
				IF fbRequest.SendJsonDomRequest(sUri:=sUri, fbClient:=fbClient, eRequestType:=eRequestType, fbJson, fbHeader) THEN				
					state := 2;
					reqCount:=reqCount+1;
				END_IF
			END_IF
		ELSE
			IF bDynamicContent THEN 
				//sSndContent := CONCAT('Test', UDINT_TO_STRING(reqCount));
				sSndContent := UDINT_TO_STRING(reqCount);
			END_IF
			nSndContent := TO_UDINT(LEN(sSndContent));
			IF nSndContent > 0 THEN
				pSndContent := ADR(sSndContent);
			ELSE
				pSndContent := NULL;
			END_IF
			IF NOT bWithHeader THEN			
				IF fbRequest.SendRequest(sUri:=sUri, fbClient:=fbClient, eRequestType:=eRequestType, pContent:=pSndContent, nContentSize:=nSndContent, 0) THEN				
					state := 2;
					reqCount:=reqCount+1;
				END_IF
			ELSE  
				IF fbRequest.SendRequest(sUri:=sUri, fbClient:=fbClient, eRequestType:=eRequestType, pContent:=pSndContent, nContentSize:=nSndContent, fbHeader) THEN				
					state := 2;
					reqCount:=reqCount+1;
				END_IF
			END_IF
		END_IF
	END_IF
2:
	IF NOT fbRequest.bBusy THEN
			IF NOT fbRequest.bError THEN
				jsonDoc := fbRequest.GetJsonDomContent(fbJson);				
				IF  jsonDoc <> 0 THEN
					bJsonRes := TRUE;
					fbJson.CopyDocument(sJson, SIZEOF(sJson)-1);
				ELSE
					bJsonRes := FALSE;
				END_IF					
				fbRequest.GetContent(pContent:=ADR(sContent), nContentSize:=SIZEOF(sContent)-1, bSetNullTermination:=TRUE);	
				fbRequest.GetHeaderField('server', ADR(sServer), SIZEOF(sServer));
					
				IF fbRequest.nStatusCode >= 200 AND fbRequest.nStatusCode < 300 THEN
					IF bDynamicContent OR bJson THEN
						IF bJsonRes THEN
						(* expected: '{"args":{},"data":"xxx(x=reqCount)","files":{},"form":{},"headers":{"x-forwarded-proto":"https","host":"postman-echo.com","content-length":"5","accept-encoding":"identity","content-type":"text/html; charset=UTF-8","user-agent":"TcHttpClient","x-forwarded-port":"443"},"json":null,"url":"https://postman-echo.com/post"}'*)								 								
							IF fbJson.HasMember(jsonDoc, 'data')  THEN
								jsonVal := fbJson.FindMember(jsonDoc, 'data');
								resVal:=fbJson.GetString(jsonVal);
								IF STRING_TO_UDINT(resVal)+1 = reqCount THEN
									valOkCount:=valOkCount+1;
								ELSE
									invResValCount:=invResValCount+1;
								END_IF
							ELSIF fbJson.HasMember(jsonDoc, 'userId')  THEN
								jsonVal := fbJson.FindMember(jsonDoc, 'userId');
								IF fbJson.GetUint(jsonVal)+1 = reqCount THEN
									valOkCount:=valOkCount+1;
								ELSE
									invResValCount:=invResValCount+1;
								END_IF
							ELSE 
								invResCount:=invResCount+1;	
							END_IF
						ELSE
							invResCount:=invResCount+1;
						END_IF
					END_IF
					nResCnt:=nResCnt+1;
				ELSE
					nErrCnt1:=nErrCnt1+1;					
				END_IF				
			ELSE
				nErrCnt2:=nErrCnt2+1;
			END_IF
			state :=1;				
	END_IF  	
END_CASE
fbClient.Execute();

END_FUNCTION_BLOCK
